PROGRAM ledLogic
VAR
	// LEDs
	ledLevel0 : BOOL := FALSE;	// Set target floor to base floor
	ledLevel1 : BOOL := FALSE;	// Set target floor to first floor
	ledLevel2 : BOOL := FALSE;	// Set target floor to seocnd floor
	ledLiftMoving : BOOL := FALSE;
	ledDoorsOpen : BOOL := FALSE;
END_VAR

// Turn of leds
IF CheckIfAtFloor() THEN
	IF GVL.liftOperation = FALSE THEN
		// Turn off buttom ledLevels
		ledLevel0 := FALSE;
		ledLevel1 := FALSE;
		ledLevel2 := FALSE;
		ledDoorsOpen := TRUE;
	END_IF
END_IF

// Turn on door LED
IF GVL.callLevel0 THEN
	ledLevel0 := TRUE;
END_IF

// Turn on door LED
IF GVL.callLevel1 THEN
	ledLevel1 := TRUE;
END_IF

// Turn on door LED
IF GVL.callLevel2 THEN
	ledLevel2 := TRUE;
END_IF

// Turn on door LED
IF GVL.liftMoving THEN
	ledLiftMoving := TRUE;
ELSE ledLiftMoving := FALSE;
END_IF

// Turn on door LED
IF GVL.openDoor THEN
	ledDoorsOpen := TRUE;
ELSE ledDoorsOpen := FALSE;
END_IF

END_PROGRAM

(* stored: Version 1.1.0.1, ProductVersion 3.1.4024.12
   POU ledLogic: Id {1b66c6d5-e132-4dd6-bb1d-63572541cf58}, SpecialFunc None *)
